// Struckig
// Copyright (C) 2022 Stefan Besler

// This program is free software: you can redistribute it and/or modify
// it under the terms of the GNU General Public License as published by
// the Free Software Foundation, either version 3 of the License, or
// (at your option) any later version.

// This program is distributed in the hope that it will be useful,
// but WITHOUT ANY WARRANTY; without even the implied warranty of
// MERCHANTABILITY or FITNESS FOR A PARTICULAR PURPOSE.  See the
// GNU General Public License for more details.
//
// You should have received a copy of the GNU General Public License
// along with THIS PROGRAM.  IF NOT, see <http://www.gnu.org/licenses/>.
/// The state Profile for position, velocity, acceleration and jerk for a single DoF
/// A single-dof kinematic profile with position, velocity, acceleration and jerk
{attribute 'hide'}
FUNCTION_BLOCK ProfileDesc
VAR_INPUT
  Limits : ReachedLimits;
  Direction : ProfileDirection;
  ControlSigns : ProfileControlSigns;
  
  t, t_sum, j : ARRAY[0..6] OF LREAL;
  a, v, p : ARRAY[0..7] OF LREAL;

  pf, vf, af : LREAL; //! Target (final) kinematic state
  Brake, Accel : BrakeProfile; //! Brake sub-profiles
END_VAR

METHOD Bound : ProfileBound
VAR_INPUT
END_VAR
VAR
  i : INT;
  t_current_sum : LREAL;
END_VAR
Bound.Minimum := Constants.Infinity;
Bound.Maximum := -Constants.Infinity;

IF Brake.Duration > 0.0
THEN
  IF (Brake.t[0] > 0.0)
  THEN
    CheckStepForBound(0.0, Brake.t[0], Brake.p[0], Brake.v[0], Brake.a[0], Brake.j[0], Bound);
  
    IF (Brake.t[1] > 0.0) 
    THEN
      CheckStepForBound(Brake.t[0], Brake.t[1], Brake.p[1], Brake.v[1], Brake.a[1], Brake.j[1], Bound);
      
      IF (Brake.t[2] > 0.0)
      THEN
        CheckStepForBound(Brake.t[0] + Brake.t[1], Brake.t[2], Brake.p[2], Brake.v[2], Brake.a[2], Brake.j[2], Bound);
      END_IF
    END_IF
  END_IF
END_IF

t_current_sum := 0;        
FOR i:=0 TO 6
DO
  IF i > 0
  THEN
    t_current_sum := t_sum[i-1];
	END_IF
  
  CheckStepForBound(t_current_sum + Brake.Duration, t[i], p[i], v[i], a[i], j[i], Bound);
END_FOR 

IF (pf < Bound.Minimum)
THEN
  Bound.Minimum := pf;
  Bound.Tmin := t_sum[6] + Brake.Duration;
END_IF 


IF (pf > Bound.Maximum) 
THEN
  Bound.Maximum := pf;
  Bound.Tmax := t_sum[6] + Brake.Duration;
END_IF
END_METHOD

METHOD CheckBound : BOOL
VAR_INPUT
  t_ext, t_sum, t, p, v, a, j : LREAL;
END_VAR
VAR_IN_OUT
  b : ProfileBound;     
END_VAR
VAR
  p_ext, v_Ext, a_ext : LREAL;
END_VAR
IF (0 < t_ext AND_THEN t_ext < t)
THEN
  Integrate(t_ext, p, v, a, j, p:=p_ext, v:=v_ext, a:=a_ext);
  IF (a_ext > 0 AND_THEN p_ext < b.Minimum)
  THEN
    b.Minimum := p_ext;
    b.Tmin := t_sum + t_ext;
   ELSIF (a_ext < 0 AND_THEN p_ext > b.Maximum) 
   THEN
    b.Maximum := p_ext;
    b.Tmax := t_sum + t_ext; 
  END_IF
END_IF
END_METHOD

/// For velocity interface
METHOD CheckForFirstOrder : BOOL
VAR_INPUT
  controlSigns : ProfileControlSigns;
  limits : ReachedLimits;  
  vUp : LREAL;
END_VAR
VAR
  i : INT;
  vUppLim : LREAL;
  vLowLim : LREAL;
  v_a_zero : LREAL;
END_VAR
// ReachedLimits::VEL
IF t[3] < 0.0
THEN
  RETURN;
END_IF

t_sum[0] := 0;
t_sum[1] := 0;
t_sum[2] := 0;
t_sum[3] := t[3];
t_sum[4] := t[3];
t_sum[5] := t[3];
t_sum[6] := t[3];

IF t_sum[6] > Constants.Tmax // For numerical reasons, is that needed?}
THEN
  RETURN;        
END_IF

j[0] := 0;
j[1] := 0;
j[2] := 0;
j[3] := 0;
j[4] := 0;
j[5] := 0;
j[6] := 0;

a[0] := 0;
a[1] := 0;
a[2] := 0;
a[3] := 0;
a[4] := 0;
a[5] := 0;
a[6] := 0;
a[7] := af;

v[0] := 0;
v[1] := 0;
v[2] := 0;
v[3] := SEL(t[3] > 0, 0, vUp);
v[4] := 0;
v[5] := 0;
v[6] := 0;
v[7] := vf;

FOR i:= 0 TO 6 
DO
  p[i+1] := p[i] + t[i] * (v[i] + t[i] * a[i] / 2);
END_FOR

THIS^.Direction := SEL(vUp > 0, ProfileDirection.Down, ProfileDirection.Up);
THIS^.ControlSigns := controlSigns;
THIS^.Limits := limits;

// Velocity limit can be broken in the beginning if both initial velocity and acceleration are too high
CheckForFirstOrder := ABS(p[7] - pf) < Constants.PositionPrecision;
END_METHOD

/// For velocity interface
METHOD CheckForFirstOrderWithTiming : BOOL
VAR_INPUT
  controlSigns : ProfileControlSigns;
  limits : ReachedLimits;  
  vUp : LREAL;
END_VAR
VAR
  i : INT;
  aUppLim : LREAL;
  aLowLim : LREAL;
END_VAR
CheckForFirstOrderWithTiming := CheckForFirstOrder(controlSigns, limits, vUp); // AND_THEN (ABS(t[6] - tf) < t_precision);
END_METHOD

/// For velocity interface
METHOD CheckForFirstOrderWithTiming2 : BOOL
VAR_INPUT
  controlSigns : ProfileControlSigns;
  limits : ReachedLimits;  
  tf : LREAL;
  vUp : LREAL;
  vMax, vMin : LREAL;
END_VAR
CheckForFirstOrderWithTiming2 :=
  (vMin - Constants.VelocityEpsilon < vUp)
  AND_THEN (vUp < vMax + Constants.VelocityEpsilon)
  AND_THEN CheckForFirstOrderWithTiming(controlSigns, limits, vUp);
END_METHOD

/// For velocity interface
METHOD CheckForSecondOrder : BOOL
VAR_INPUT
  controlSigns : ProfileControlSigns;
  limits : ReachedLimits;  
  aUp, aDown : LREAL;
  vMax, vMin : LREAL;
END_VAR
VAR
  i : INT;
  vUppLim : LREAL;
  vLowLim : LREAL;
  v_a_zero : LREAL;
END_VAR
// ReachedLimits::ACC0
IF t[0] < 0.0
THEN
  RETURN;
END_IF

t_sum[0] := t[0];
FOR i:=0 TO 5
DO
  IF (t[i+1] < 0)
  THEN
    RETURN;
  END_IF
  
  t_sum[i+1] := t_sum[i] + t[i+1];  
END_FOR

IF t_sum[6] > Constants.Tmax // For numerical reasons, is that needed?}
THEN
  RETURN;        
END_IF

j[0] := 0;
j[1] := 0;
j[2] := 0;
j[3] := 0;
j[4] := 0;
j[5] := 0;
j[6] := 0;

IF controlSigns = ProfileControlSigns.Uddu
THEN
  a[0] := SEL(t[0] > 0, 0, aUp);
  a[1] := 0;
  a[2] := SEL(t[2] > 0, 0, aDown);
  a[3] := 0;
  a[4] := SEL(t[4] > 0, 0, aDown);
  a[5] := 0;
  a[6] := SEL(t[6] > 0, 0, aUp);
  a[7] := af;
ELSE
  a[0] := SEL(t[0] > 0, 0, aUp);
  a[1] := 0;
  a[2] := SEL(t[2] > 0, 0, aDown);
  a[3] := 0;
  a[4] := SEL(t[4] > 0, 0, aUp);
  a[5] := 0;
  a[6] := SEL(t[6] > 0, 0, aDown);
  a[7] := af;
END_IF

direction := SEL(vMax > 0, ProfileDirection.Down, ProfileDirection.Up);
vUppLim := SEL(direction = ProfileDirection.Up, vMin, vMax) + Constants.VelocityEpsilon;
vLowLim := SEL(direction = ProfileDirection.Up, vMax, vMin) - Constants.VelocityEpsilon;

FOR i:= 0 TO 6 
DO
  v[i+1] := v[i] + t[i] * a[i];
  p[i+1] := p[i] + t[i] * (v[i] + t[i] * a[i] / 2);
END_FOR


THIS^.ControlSigns := controlSigns;
THIS^.Limits := limits;

// Velocity limit can be broken in the beginning if both initial velocity and acceleration are too high
CheckForSecondOrder := ABS(p[7] - pf) < Constants.PositionPrecision AND_THEN ABS(v[7] - vf) < Constants.VelocityPrecision
    AND_THEN v[2] <= vUppLim AND_THEN v[3] <= vUppLim AND_THEN v[4] <= vUppLim AND_THEN v[5] <= vUppLim AND_THEN v[6] <= vUppLim
    AND_THEN v[2] >= vLowLim AND_THEN v[3] >= vLowLim AND_THEN v[4] >= vLowLim AND_THEN v[5] >= vLowLim AND_THEN v[6] >= vLowLim;
END_METHOD

/// For velocity interface
METHOD CheckForSecondOrderVelocity : BOOL
VAR_INPUT
  controlSigns : ProfileControlSigns;
  limits : ReachedLimits;  
  aUp : LREAL;
END_VAR
VAR
  i : INT;
  aUppLim : LREAL;
  aLowLim : LREAL;
END_VAR
// ReachedLimits::ACC0
IF t[1] < 0.0
THEN
  RETURN;
END_IF

t_sum[0] := 0;
t_sum[1] := t[1];
t_sum[2] := t[1];
t_sum[3] := t[1];
t_sum[4] := t[1];
t_sum[5] := t[1];
t_sum[6] := t[1];

// For numerical reasons, is that needed?
IF t_sum[6] > Constants.Tmax
THEN
  RETURN;
END_IF


j[0] := 0;
j[1] := 0;
j[2] := 0;
j[3] := 0;
j[4] := 0;
j[5] := 0;
j[6] := 0;

a[0] := 0;
a[1] := aUp;
a[2] := 0;
a[3] := 0;
a[4] := 0;
a[5] := 0;
a[6] := 0;
a[7] := THIS^.af;

FOR i:=0 TO 6
DO
  v[i+1] := v[i] + t[i] * a[i];
  p[i+1] := p[i] + t[i] * (v[i] + t[i] * a[i] / 2);
END_FOR

THIS^.ControlSigns := controlSigns;
THIS^.Limits := limits;
THIS^.Direction := SEL(aUp > 0, ProfileDirection.Down, ProfileDirection.Up);

// Velocity limit can be broken in the beginning if both initial velocity and acceleration are too high
CheckForSecondOrderVelocity := ABS(v[6] - vf) < Constants.VelocityPrecision;
END_METHOD

/// For velocity interface
METHOD CheckForSecondOrderVelocityWithTiming : BOOL
VAR_INPUT
  controlSigns : ProfileControlSigns;
  limits : ReachedLimits;  
  aUp : LREAL;
END_VAR
CheckForSecondOrderVelocityWithTiming := CheckForSecondOrderVelocity(controlSigns, limits, aUp); // AND_THEN (ABS(t[6] - tf) < t_precision);
END_METHOD

/// For velocity interface
METHOD CheckForSecondOrderVelocityWithTiming2 : BOOL
VAR_INPUT
  controlSigns : ProfileControlSigns;
  limits : ReachedLimits;  
  tf : LREAL;
  aUp : LREAL;
  aMax : LREAL;
  aMin : LREAL;
END_VAR
CheckForSecondOrderVelocityWithTiming2 :=
 (aMin - Constants.AccelerationEpsilon < aUp)
 AND_THEN (aUp < aMax + Constants.AccelerationEpsilon)
 AND_THEN CheckForSecondOrderVelocityWithTiming(controlSigns, limits, aUp); // AND_THEN (ABS(t[6] - tf) < t_precision);
END_METHOD

/// For velocity interface
METHOD CheckForSecondOrderWithTiming : BOOL
VAR_INPUT
  controlSigns : ProfileControlSigns;
  limits : ReachedLimits;  
  tf : LREAL;
  aUp, aDown : LREAL;
  vMax, vMin : LREAL;
END_VAR
CheckForSecondOrderWithTiming := CheckForSecondOrder(controlSigns, limits, aUp, aDown, vMax, vMin);
END_METHOD

/// For velocity interface
METHOD CheckForSecondOrderWithTiming2 : BOOL
VAR_INPUT
  controlSigns : ProfileControlSigns;
  limits : ReachedLimits;  
  tf : LREAL;
  aUp, aDown : LREAL;
  vMax, vMin : LREAL;
  aMax, aMin : LREAL;  
END_VAR
CheckForSecondOrderWithTiming2 := 
    (aMin - Constants.AccelerationEpsilon < aUp)
    AND_THEN (aUp < aMax + Constants.AccelerationEpsilon)
    AND_THEN (aMin - Constants.AccelerationEpsilon < aDown)
    AND_THEN (aDown < aMax + Constants.AccelerationEpsilon)
    AND_THEN CheckForSecondOrderWithTiming(controlSigns, limits,tf, aUp, aDown, vMax, vMin);
END_METHOD

/// For velocity interface
METHOD CheckForVelocity : BOOL
VAR_INPUT
  controlSigns : ProfileControlSigns;
  limits : ReachedLimits;  
  jf : LREAL;
  aMax : LREAL;
  aMin : LREAL;  
END_VAR
VAR
  i : INT;
  aUppLim : LREAL;
  aLowLim : LREAL;
END_VAR
IF (t[0] < 0)
THEN
  RETURN;
END_IF

t_sum[0] := t[0];
FOR i:=0 TO 5
DO
  IF (t[i+1] < 0)
  THEN
    RETURN;
  END_IF
  
  t_sum[i+1] := t_sum[i] + t[i+1];
END_FOR


IF limits = ReachedLimits.Acc0
THEN
  IF t[1] < Constants.DoubleEpsilon
  THEN
    RETURN;
  END_IF
END_IF


IF t_sum[6] > Constants.Tmax // For numerical reasons, is that needed?}
THEN
  RETURN;        
END_IF

IF controlSigns = ProfileControlSigns.Uddu
THEN
  j[0] := SEL(t[0] > 0, 0, jf);
  j[1] := 0;
  j[2] := SEL(t[2] > 0, 0, -jf);
  j[3] := 0;
  j[4] := SEL(t[4] > 0, 0, -jf);
  j[5] := 0;
  j[6] := SEL(t[6] > 0, 0, jf);          
ELSE
  j[0] := SEL(t[0] > 0, 0, jf);
  j[1] := 0;
  j[2] := SEL(t[2] > 0, 0, -jf);
  j[3] := 0;
  j[4] := SEL(t[4] > 0, 0, jf);
  j[5] := 0;
  j[6] := SEL(t[6] > 0, 0, -jf); 
END_IF


FOR i:=0 TO 6
DO
  a[i+1] := a[i] + t[i] * j[i];
  v[i+1] := v[i] + t[i] * (a[i] + t[i] * j[i] / 2);
  p[i+1] := p[i] + t[i] * (v[i] + t[i] * (a[i] / 2 + t[i] * j[i] / 6));        
END_FOR

      
THIS^.ControlSigns := controlSigns;
THIS^.Limits := limits;

aUppLim := SEL((aMax > 0), aMin, aMax) + 5E-12;
aLowLim := SEL((aMax > 0), aMax, aMin) - 5E-12;

// Velocity limit can be broken in the beginning if both initial velocity and acceleration are too high
CheckForVelocity := ABS(v[7] - vf) < Constants.VelocityPrecision
    AND_THEN ABS(a[7] - af) < Constants.AccelerationPrecision // This is not really needed, but we want to double check
    AND_THEN a[1] >= aLowLim AND_THEN a[3] >= aLowLim AND_THEN a[5] >= aLowLim
    AND_THEN a[1] <= aUppLim AND_THEN a[3] <= aUppLim AND_THEN a[5] <= aUppLim;
END_METHOD

/// For velocity interface
METHOD CheckForVelocityWithTiming : BOOL
VAR_INPUT
  controlSigns : ProfileControlSigns;
  limits : ReachedLimits;  
  jf : LREAL;
  aMax : LREAL;
  aMin : LREAL;  
  jMax : LREAL;  
END_VAR
// Time doesn't need to be checked as every profile has a: tf - ... equation
CheckForVelocityWithTiming := (ABS(jf) < ABS(jMax) + Constants.JerkEpsilon) AND_THEN CheckForVelocity(controlSigns, limits, jf, aMax, aMin);
END_METHOD

METHOD CheckStepForBound : BOOL
VAR_INPUT
  t_sum, t, p, v, a, j : LREAL;
END_VAR
VAR_IN_OUT
  b : ProfileBound;  
END_VAR
VAR
  d, d_sqrt : LREAL;
END_VAR
IF (p < b.Minimum)
THEN 
  b.Minimum := p;
  b.Tmin := t_sum;
END_IF

IF (p > b.Maximum)
THEN 
  b.Maximum := p;
  b.Tmax := t_sum;
END_IF

IF (j <> 0) 
THEN
  d := a * a - 2 * j * v;
  IF (ABS(d) < Constants.DoubleEpsilon)
  THEN
    CheckBound(-a / j, t_sum, t, p, v, a, j, b:=b);
   ELSIF (d > 0) 
   THEN
    d_sqrt := SQRT(d);
    CheckBound((-a - D_sqrt) / j, t_sum, t, p, v, a, j, b:=b);
    CheckBound((-a + D_sqrt) / j, t_sum, t, p, v, a, j, b:=b);           
  END_IF
END_IF
END_METHOD

/// For position interface
METHOD CheckVel : BOOL
VAR_INPUT
  controlSigns : ProfileControlSigns;    
  limits : ReachedLimits;
  jf : LREAL;
  vMax : LREAL;
  vMin : LREAL;  
  aMax : LREAL;
  aMin : LREAL;
  setLimits : BOOL;
END_VAR
VAR
  i : INT;
  v_a_zero : LREAL;
  vUppLim, vLowLim : LREAL;  
  aUppLim, aLowLim : LREAL;
END_VAR
IF (t[0] < 0) 
THEN
  RETURN;
END_IF

t_sum[0] := t[0];
FOR i:=0 TO 5
DO
  IF (t[i+1] < 0)
  THEN
    RETURN;
  END_IF
  
  t_sum[i+1] := t_sum[i] + t[i+1];  
END_FOR

IF limits = ReachedLimits.Acc0Acc1Vel OR_ELSE limits = ReachedLimits.Acc0Vel OR_ELSE limits = ReachedLimits.Acc1Vel OR_ELSE limits = ReachedLimits.Vel THEN
  IF (t[3] < Constants.DoubleEpsilon) 
  THEN
    RETURN;                    
  END_IF
END_IF

IF limits = ReachedLimits.Acc0 OR_ELSE limits = ReachedLimits.Acc0Acc1
THEN
  IF (t[1] < Constants.DoubleEpsilon) 
  THEN
    RETURN;                    
  END_IF
END_IF

IF limits = ReachedLimits.Acc1 OR_ELSE limits = ReachedLimits.Acc0Acc1
THEN
  IF (t[5] < Constants.DoubleEpsilon)
  THEN
    RETURN;            
  END_IF
END_IF

IF t_sum[6] > Constants.Tmax  // For numerical reasons, is that needed?
THEN
  RETURN;        
END_IF
        
IF controlSigns = ProfileControlSigns.Uddu
THEN
  j[0] := SEL(t[0] > 0, 0, jf);
  j[1] := 0;
  j[2] := SEL(t[2] > 0, 0, -jf);
  j[3] := 0;
  j[4] := SEL(t[4] > 0, 0, -jf);
  j[5] := 0;
  j[6] := SEL(t[6] > 0, 0, jf);          
ELSE
  j[0] := SEL(t[0] > 0, 0, jf);
  j[1] := 0;
  j[2] := SEL(t[2] > 0, 0, -jf);
  j[3] := 0;
  j[4] := SEL(t[4] > 0, 0, jf);
  j[5] := 0;
  j[6] := SEL(t[6] > 0, 0, -jf); 
END_IF

vUppLim := SEL(vMax > 0, vMin, vMax) + 1E-12;
vLowLim := SEL(vMax > 0, vMax, vMin) - 1E-12;

direction := SEL(vMax > 0, ProfileDirection.Down, ProfileDirection.Up);
vUppLim := SEL(direction = ProfileDirection.Up, vMin, vMax) + Constants.VelocityEpsilon;
vLowLim := SEL(direction = ProfileDirection.Up, vMax, vMin) - Constants.VelocityEpsilon;
        
FOR i:= 0 TO 6 
DO
  a[i+1] := a[i] + t[i] * j[i];
  v[i+1] := v[i] + t[i] * (a[i] + t[i] * j[i] / 2);
  p[i+1] := p[i] + t[i] * (v[i] + t[i] * (a[i] / 2 + t[i] * j[i] / 6));

  IF limits = ReachedLimits.Acc0Acc1Vel OR_ELSE limits = ReachedLimits.Acc0Acc1 OR_ELSE limits = ReachedLimits.Acc0Vel OR_ELSE limits = ReachedLimits.Acc1Vel OR_ELSE limits = ReachedLimits.Vel
  THEN
    IF i = 2
    THEN
     a[3] := 0.0;
    END_IF
  END_IF
  
  IF setLimits
  THEN
    IF limits = ReachedLimits.Acc1
    THEN
      IF i = 2
      THEN
        a[3] := aMin;
      END_IF
    ELSIF limits = ReachedLimits.Acc0Acc1
    THEN
      CASE i
      OF
      0: a[1] := aMax;
      4: a[5] := aMin;
      END_CASE  
    END_IF
  END_IF
  
  IF (i > 1 AND_THEN a[i+1] * a[i] < -Constants.DoubleEpsilon) 
  THEN
    v_a_zero := v[i] - (a[i] * a[i]) / (2 * j[i]);
    IF (v_a_zero > vUppLim OR_ELSE v_a_zero < vLowLim)
    THEN
      RETURN;        
		END_IF
  END_IF
END_FOR


THIS^.ControlSigns := controlSigns;
THIS^.Limits := limits;

aUppLim := SEL(direction = ProfileDirection.Up, aMin, aMax) + Constants.AccelerationEpsilon;
aLowLim := SEL(direction = ProfileDirection.Up, aMax, aMin) - Constants.AccelerationEpsilon;

// Velocity limit can be broken in the beginning if both initial velocity and acceleration are too high
CheckVel := ABS(p[7] - pf) < Constants.PositionPrecision
    AND_THEN ABS(v[7] - vf) < Constants.VelocityPrecision
    AND_THEN ABS(a[7] - af) < Constants.AccelerationPrecision // This is not really needed, but we want to double check
    // AND_THEN ABS(v[3]) <= vMaxAbs AND_THEN ABS(v[4]) <= vMaxAbs AND_THEN ABS(v[5]) <= vMaxAbs AND_THEN ABS(v[6]) <= vMaxAbs
    AND_THEN a[1] >= aLowLim AND_THEN a[3] >= aLowLim AND_THEN a[5] >= aLowLim
    AND_THEN a[1] <= aUppLim AND_THEN a[3] <= aUppLim AND_THEN a[5] <= aUppLim
    AND_THEN v[3] <= vUppLim AND_THEN v[4] <= vUppLim AND_THEN v[5] <= vUppLim AND_THEN v[6] <= vUppLim
    AND_THEN v[3] >= vLowLim AND_THEN v[4] >= vLowLim AND_THEN v[5] >= vLowLim AND_THEN v[6] >= vLowLim; // this is not really needed, but we want to double check
END_METHOD

METHOD CheckWithTiming : BOOL
VAR_INPUT
  controlSigns : ProfileControlSigns;    
  limits : ReachedLimits;
  tf : LREAL;
  jf : LREAL;
  vMax : LREAL;
  vMin : LREAL;  
  aMax : LREAL;
  aMin : LREAL;  
END_VAR
// Time doesn't need to be checked as every Profile has a: tf - ... equation
CheckWithTiming := CheckVel(controlSigns, limits, jf, vMax, vMin, aMax, aMin, setLimits:=FALSE); // && (std::abs(t_sum[6] - tf) < Constants.TimePrecision)
END_METHOD

METHOD CheckWithTiming2 : BOOL
VAR_INPUT
  controlSigns : ProfileControlSigns;    
  limits : ReachedLimits;
  tf : LREAL;
  jf : LREAL;
  vMax : LREAL;
  vMin : LREAL;  
  aMax : LREAL;
  aMin : LREAL;
  jMax  : LREAL;
END_VAR
CheckWithTiming2 := (ABS(jf) < ABS(jMax) + Constants.JerkEpsilon) AND_THEN CheckWithTiming(controlSigns, limits, tf, jf, vMax, vMin, aMax, aMin);
END_METHOD

METHOD FirstStateAtPosition : BOOL
VAR_INPUT
  pt, offset : LREAL;
END_VAR
VAR_IN_OUT
  t_t, v_t, a_t : LREAL;
END_VAR
VAR
  i,h : INT;
  p_t : LREAL;
  polynom : ARRAY[0..4] OF LREAL;
  rootCount : INT;
  root : ARRAY[0..6] OF LREAL;
END_VAR
FOR i:=0 TO 6
DO
  IF ABS(p[i] - pt) < Constants.DoubleEpsilon
  THEN
    t_t := offset + SEL(i>0, 0, t_sum[i-1]);
    v_t := v[i];
    a_t := a[i];
    FirstStateAtPosition := TRUE;
    RETURN;
	END_IF
  
  IF t[i] = 0
  THEN
    CONTINUE;
	END_IF
  
  polynom[0] := j[i]/6;
  polynom[1] := a[i]*0.5;
  polynom[2] := v[i];
  polynom[3] := p[i]-pt;
  Roots.SolveCub(ADR(polynom), rootCount:=rootCount, roots:=root);
  FOR h:=0 TO rootCount
  DO
    IF(0 < root[h] AND_THEN root[h] <= t[i])
    THEN
      t_t := offset + root[h] + SEL(i>0, 0, t_sum[i-1]);
      Integrate(root[h], p[i], v[i], a[i], j[i], p_t, v_t, a_t);
      FirstStateAtPosition := TRUE;
      RETURN;      
		END_IF
  END_FOR
  
END_FOR

IF ABS(pf-pt) < Constants.Epsilon
THEN
  t_t := offset + t_sum[6];
  v_t := vf;
  a_t := af;
  FirstStateAtPosition := TRUE;
  RETURN;      
END_IF
END_METHOD

/// Set boundary values for the position interface
METHOD SetBoundary
VAR_IN_OUT CONSTANT
  profile : ProfileDesc;
END_VAR
a[0] := profile.a[0];
v[0] := profile.v[0];
p[0] := profile.p[0];
af := profile.af;
vf := profile.vf;
pf := profile.pf;
Brake := profile.Brake;
Accel := profile.Accel;
END_METHOD

/// Set boundary values for the position interface
METHOD SetBoundaryPosition
VAR_INPUT
  p0_new, v0_new, a0_new, pf_new, vf_new, af_new : LREAL;
END_VAR
a[0] := a0_new;
v[0] := v0_new;
p[0] := p0_new;
af := af_new;
vf := vf_new;
pf := pf_new;
END_METHOD

/// Set boundary values for the velocity interface
METHOD SetBoundaryVelocity
VAR_INPUT
  p0_new, v0_new, a0_new, vf_new, af_new : LREAL;
END_VAR
a[0] := a0_new;
v[0] := v0_new;
p[0] := p0_new;
af := af_new;
vf := vf_new;
END_METHOD

END_FUNCTION_BLOCK

(* stored: Version 1.1.0.1
   POU ProfileDesc: Id {1331731c-0677-4d13-b754-67c3077cc0c4}, SpecialFunc None
   Method Bound: Id {1a9ba528-afaf-4159-b889-acb983a16fac}
   Method CheckBound: Id {e3c5916b-156b-465a-87ae-6759453a325c}
   Method CheckForFirstOrder: Id {31212f13-d5a9-4742-8643-6d97fa16497a}
   Method CheckForFirstOrderWithTiming: Id {f2aee95d-8ed3-4a11-8ddd-b5d6faaeadf9}
   Method CheckForFirstOrderWithTiming2: Id {45d59201-d920-42f5-a1d0-0ce0793e419d}
   Method CheckForSecondOrder: Id {d36e3565-cce0-4f73-83f9-ec95541ce2ef}
   Method CheckForSecondOrderVelocity: Id {98d640fa-ba4c-4586-9f8c-bed3ada54742}
   Method CheckForSecondOrderVelocityWithTiming: Id {268274ba-8baf-4ee0-a4bb-6de0fd1ae36e}
   Method CheckForSecondOrderVelocityWithTiming2: Id {915c6be4-07ad-4bf6-8b4d-9b5951f90edc}
   Method CheckForSecondOrderWithTiming: Id {add5d654-e57e-4ae8-b083-d5a062804107}
   Method CheckForSecondOrderWithTiming2: Id {2570a4cc-90d1-47de-bf99-989113385597}
   Method CheckForVelocity: Id {dec39d38-9a64-41bc-99b6-6a7b67c016da}
   Method CheckForVelocityWithTiming: Id {f910072d-eaca-431a-9473-d411e940a4c7}
   Method CheckStepForBound: Id {ce8df4c2-1570-4fbc-87ab-2de79032d446}
   Method CheckVel: Id {1650deae-6774-4923-94a5-237877609b6a}
   Method CheckWithTiming: Id {a762f8df-7f20-4c45-819e-1ecbfa908ad5}
   Method CheckWithTiming2: Id {c707d6dc-e662-4300-aebc-c29e90e74532}
   Method FirstStateAtPosition: Id {0159e4a6-0809-4a0c-b389-030aa446ea6f}
   Method SetBoundary: Id {fdfe1c1e-08a5-45e1-a4af-4f8d0e84c34a}
   Method SetBoundaryPosition: Id {bcaf6cf3-3cdf-411e-b9b2-105283f26c0e}
   Method SetBoundaryVelocity: Id {5e35273a-4554-4245-bfd9-f07367ed9a5c} *)
